// TIA Portal V16 export
// export: Created 2022-09-01T09:20:33.4367343Z, ExportSetting WithDefaults, DisplayName Totally Integrated Automation Portal, DisplayVersion V16, DisplayName TIA Portal Version Control Interface, DisplayVersion V16, DisplayName TIA Portal Openness, DisplayVersion V16, DisplayName STEP 7 Professional, DisplayVersion V16, DisplayName STEP 7 Safety, DisplayVersion V16, DisplayName WinCC Advanced, DisplayVersion V16
VAR_GLOBAL   // PLC tag table "Default tag table"
   START AT %M0.0 : Bool;
   OUTPUT AT %M0.2 : Bool;
   STOP AT %M0.1 : Bool;
   MW100 AT %MW100 : Int;
END_VAR
